// Mitsubishi GX Developer project: Assignment_RotartyTransferPLC   PLC: FX2N

PROGRAM MAIN
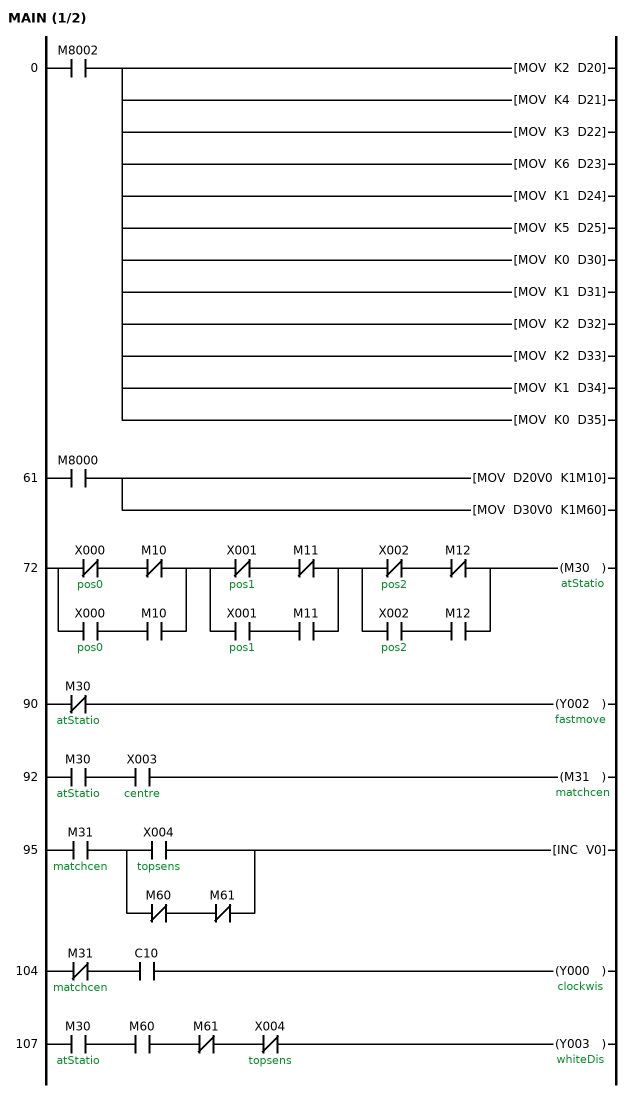
0     LD      M8002
      MOV     K2 D20
      MOV     K4 D21
      MOV     K3 D22
      MOV     K6 D23
      MOV     K1 D24
      MOV     K5 D25
      MOV     K0 D30
      MOV     K1 D31
      MOV     K2 D32
      MOV     K2 D33
      MOV     K1 D34
      MOV     K0 D35
61    LD      M8000
      MOV     D20V0 K1M10
      MOV     D30V0 K1M60
72    LDI     X000  ; pos0
      ANI     M10
      LD      X000  ; pos0
      AND     M10
      ORB
      LDI     X001  ; pos1
      ANI     M11
      LD      X001  ; pos1
      AND     M11
      ORB
      ANB
      LDI     X002  ; pos2
      ANI     M12
      LD      X002  ; pos2
      AND     M12
      ORB
      ANB
      OUT     M30  ; atStatio
90    LDI     M30  ; atStatio
      OUT     Y002  ; fastmove
92    LD      M30  ; atStatio
      AND     X003  ; centre
      OUT     M31  ; matchcen
95    LD      M31  ; matchcen
      LD      X004  ; topsens
      LDI     M60
      ANI     M61
      ORB
      ANB
      INC     V0
104   LDI     M31  ; matchcen
      AND     C10
      OUT     Y000  ; clockwis
107   LD      M30  ; atStatio
      AND     M60
      ANI     M61
      ANI     X004  ; topsens
      OUT     Y003  ; whiteDis
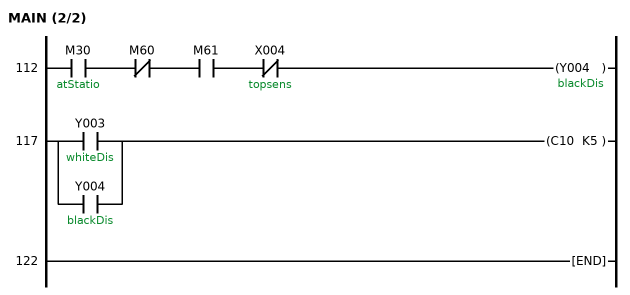
112   LD      M30  ; atStatio
      ANI     M60
      AND     M61
      ANI     X004  ; topsens
      OUT     Y004  ; blackDis
117   LD      Y003  ; whiteDis
      OR      Y004  ; blackDis
      OUT     C10 K5
122   END
END_PROGRAM

// device comments not shown above
X005  ; bottsens
X006  ; whitetop
X007  ; whitebot
X010  ; emergst
X011  ; start
Y001  ; anticlks
Y005  ; Alarm
